INTERFACE I_LoadCell

PROPERTY fActWeight : REAL
GET
END_GET
END_PROPERTY

METHOD NetMode : BOOL
VAR_INPUT
END_VAR
END_METHOD

METHOD Set_Zero : BOOL
VAR_INPUT
END_VAR
END_METHOD

PROPERTY Status : REAL
GET
END_GET
END_PROPERTY

END_INTERFACE

(* stored: Version 1.1.0.1, ProductVersion 3.1.4024.12
   Itf I_LoadCell: Id {dcfb5ceb-bdb5-4814-9d6d-fd5a46ed26c5}
   Property fActWeight: Id {3246cbd0-62f1-4573-91fe-b4fcd79dbb51}
   Get Get: Id {a889edbf-fe4c-43a8-bb64-73f6a4c75947}
   Method NetMode: Id {e062cd53-9e9c-4895-9326-952c3527d8ff}
   Method Set_Zero: Id {290b437b-6baa-42d4-af62-52c1705ca53f}
   Property Status: Id {e972a264-a2e5-4093-bf94-858432a80511}
   Get Get: Id {096fc1b9-0821-44f9-a870-2eaa740e860f} *)
